Universal Robots PolyScope program: Assignment.urp

Program Assignment (installation=assignment directory=/home/mtrn4230/ursim-5.10.0.106288/programs createdIn=5.10.0.106288 lastSavedIn=5.10.0.106288 robotSerialNumber=20195599999)
Calibrated DH parameters: a=[0, -0.425, -0.3922, 0, 0, 0]; d=[0.1625, 0, 0, 0.1333, 0.0997, 0.0996]; alpha=[1.570796, 0, 0, 1.570796, -1.570796, 0]; deltaTheta=[0, 0, 0, 0, 0, 0]
Robot Program (runOnlyOnce=false)
  SuppressedNode
    Popup Message (haltProgram=false message=EDLYN LIEW L inputType=Text)
  LETTERS := [5,4,13,25,14,27,12,9,5,23,27,12]
  num_letters := 12
  counter := 0
  MoveJ speed 60 deg/s, acceleration 80 deg/s^2 (useActiveTCP=true) feature=letter_start
    Waypoint start_corner: TCP in base x=-509.831 y=-90.3 z=70 mm, rx=2.2214 ry=2.2214 rz=0 rad; joints [-4.875, -57.642, 121.444, -153.801, -90, -4.875] deg; feature pose in base x=-509.831 y=-90.3 z=70 mm, rx=2.2214 ry=2.2214 rz=0 rad
    'start height: 70mm'
  MoveJ speed 60 deg/s, acceleration 80 deg/s^2 (useActiveTCP=true) feature=letter_start
    curr_pos := pose_trans(pose_sub(get_actual_tcp_pose(),letter_start), p[0,0,0,0,0,0])
    Loop While (checkContinuously=false) expression=counter<num_letters
      Switch expression=LETTERS[counter]
        Case (caseValue=1)
          'a'
        Case (caseValue=2)
          'b'
        Case (caseValue=3)
          'c'
        Case (caseValue=4)
          'd'
          Wait Sleep waitTime=1
          MoveJ speed 60 deg/s, acceleration 80 deg/s^2 (useActiveTCP=true) feature=letter_start
            curr_pos := pose_trans(curr_pos, p[0.65/100,0,0,0,0,0])
            Popup Message (haltProgram=false inputType=Variable) variable=curr_pos
            Waypoint Waypoint (Variable): variable=curr_pos
          MoveL speed 250 mm/s, acceleration 1200 mm/s^2 (useActiveTCP=true) feature=letter_start
            Call move_down
            curr_pos := pose_trans(curr_pos, p[0,2/100,0,0,0,0])
            Popup Message (haltProgram=false inputType=Variable) variable=curr_pos
            Waypoint Waypoint (Variable): variable=curr_pos
            end_circle := curr_pos
            Popup Message (haltProgram=false inputType=Variable) variable=curr_pos
            Call move_up
            curr_pos := pose_trans(curr_pos, p[0,-2/100,0,0,0,0])
            Call move_down
            Popup Message (haltProgram=false inputType=Variable) variable=curr_pos
          MoveP speed 250 mm/s, acceleration 1200 mm/s^2 (blendRadius=0.025 useActiveTCP=true) feature=letter_start
            Waypoint Waypoint (Variable): variable=curr_pos
            circle_via := pose_trans(curr_pos, p[1.35/100,1/100,0,0,0,0])
            CircleMove (OrientationMode=UNCONSTRAINED)
              Waypoint Waypoint (Variable): variable=circle_via
              Waypoint Waypoint (Variable): variable=end_circle
          MoveL speed 250 mm/s, acceleration 1200 mm/s^2 (useActiveTCP=true) feature=letter_start
            curr_pos := end_circle
            Waypoint Waypoint (Variable): variable=curr_pos
            Call move_up
            curr_pos := pose_trans(curr_pos, p[1.35/100,-2/100,0,0,0,0])
        Case (caseValue=5)
          'e'
          Wait Sleep waitTime=1
          MoveL speed 250 mm/s, acceleration 1200 mm/s^2 (useActiveTCP=true) feature=letter_start
            Call move_down
            curr_pos := pose_trans(curr_pos, p[0,2/100,0,0,0,0])
            Waypoint Waypoint (Variable): variable=curr_pos
            SuppressedNode
              Popup Message (haltProgram=false inputType=Variable) variable=curr_pos
            curr_pos := pose_trans(curr_pos, p[1/100,0,0,0,0,0])
            SuppressedNode
              Popup Message (haltProgram=false inputType=Variable) variable=curr_pos
            Waypoint Waypoint (Variable): variable=curr_pos
            Call move_up
            SuppressedNode
              Popup Message (haltProgram=false inputType=Variable) variable=curr_pos
            curr_pos := pose_trans( curr_pos,p[-1/100,-2/100,0,0,0,0])
            SuppressedNode
              Popup Message (haltProgram=false inputType=Variable) variable=curr_pos
            Waypoint Waypoint (Variable): variable=curr_pos
            Call move_down
            curr_pos := pose_trans(curr_pos, p[1.1/100,0,0,0,0,0])
            Waypoint Waypoint (Variable): variable=curr_pos
            Call move_up
            curr_pos := pose_trans(curr_pos,p[-1.1/100,0.9/100,0,0,0,0])
            Waypoint Waypoint (Variable): variable=curr_pos
            Call move_down
            curr_pos := pose_trans(curr_pos, p[1/100,0,0,0,0,0])
            Waypoint Waypoint (Variable): variable=curr_pos
            Popup Message (haltProgram=false inputType=Variable) variable=curr_pos
            Call move_up
            curr_pos := pose_trans(curr_pos, p[0.1/100,-0.9/100,0,0,0,0])
            Waypoint Waypoint (Variable): variable=curr_pos
            Popup Message (haltProgram=false inputType=Variable) variable=curr_pos
        Case (caseValue=6)
          'f'
        Case (caseValue=7)
          'g'
        Case (caseValue=8)
          'h'
        Case (caseValue=9)
          'i'
        Case (caseValue=10)
          'j'
        Case (caseValue=11)
          'k'
        Case (caseValue=12)
          'l'
          Wait Sleep waitTime=1
          MoveL speed 250 mm/s, acceleration 1200 mm/s^2 (useActiveTCP=true) feature=letter_start
            curr_pos := pose_trans(curr_pos, p[0.7/100,0,0,0,0,0])
            Waypoint Waypoint (Variable): variable=curr_pos
            Call move_down
            curr_pos := pose_trans(curr_pos, p[0,2/100,0,0,0,0])
            Waypoint Waypoint (Variable): variable=curr_pos
            curr_pos := pose_trans(curr_pos, p[1/100,0,0,0,0,0])
            Waypoint Waypoint (Variable): variable=curr_pos
            Call move_up
            curr_pos := pose_trans(curr_pos,p[0.2/100,-2/100,0,0,0,0])
        Case (caseValue=13)
          'm'
        Case (caseValue=14)
          'n'
          Wait Sleep waitTime=1
          MoveJ speed 60 deg/s, acceleration 80 deg/s^2 (useActiveTCP=true) feature=letter_start
            curr_pos := pose_trans(curr_pos, p[0.3,0,0,0,0,0])
            Waypoint Waypoint (Variable): variable=curr_pos
            Call move_down
            curr_pos := pose_trans(curr_pos, p[0,2/100,0,0,0,0])
            Waypoint Waypoint (Variable): variable=curr_pos
            Call move_up
            curr_pos := pose_trans(curr_pos, p[0,-2/100,0,0,0,0])
            Waypoint Waypoint (Variable): variable=curr_pos
            Call move_down
            curr_pos := pose_trans(curr_pos, p[1.25/100,2/100,0,0,0,0])
            Waypoint Waypoint (Variable): variable=curr_pos
            Call move_up
            curr_pos := pose_trans(curr_pos, p[0,-2/100,0,0,0,0])
            Waypoint Waypoint (Variable): variable=curr_pos
            Call move_down
            curr_pos := pose_trans(curr_pos, p[0,2/100,0,0,0,0])
            Waypoint Waypoint (Variable): variable=curr_pos
            Call move_up
            curr_pos := pose_trans(curr_pos, p[0.2/100,-2/100,0,0,0,0])
        Case (caseValue=15)
          'o'
        Case (caseValue=16)
          'p'
        Case (caseValue=17)
          'q'
        Case (caseValue=18)
          'r'
        Case (caseValue=19)
          's'
        Case (caseValue=20)
          't'
        Case (caseValue=21)
          'u'
        Case (caseValue=22)
          'v'
        Case (caseValue=23)
          'w'
        Case (caseValue=24)
          'x'
        Case (caseValue=25)
          'y'
          Wait Sleep waitTime=1
          MoveJ speed 60 deg/s, acceleration 80 deg/s^2 (useActiveTCP=true) feature=letter_start
            curr_pos := pose_trans(curr_pos, p[0.3/100,0,0,0,0,0])
            Waypoint Waypoint (Variable): variable=curr_pos
            Call move_down
            curr_pos := pose_trans(curr_pos, p[0.8/100,1.3/100,0,0,0,0])
            Waypoint Waypoint (Variable): variable=curr_pos
            Call move_up
            curr_pos := pose_trans(curr_pos, p[0.8/100,-1.3/100,0,0,0,0])
            Waypoint Waypoint (Variable): variable=curr_pos
            Call move_down
            curr_pos := pose_trans(curr_pos, p[-0.8/100,1.3/100,0,0,0,0])
            Waypoint Waypoint (Variable): variable=curr_pos
            curr_pos := pose_trans(curr_pos, p[0,0.8/100,0,0,0,0])
            Waypoint Waypoint (Variable): variable=curr_pos
            Call move_up
            curr_pos := pose_trans(curr_pos, p[1/100,-2/100,0,0,0,0])
        Case (caseValue=26)
          'z'
        Case (caseValue=27)
          'space'
          Wait Sleep waitTime=1
          curr_pos := pose_trans(curr_pos, p[2.2/100,0,0,0,0,0])
      counter := counter+1
  MoveJ speed 60 deg/s, acceleration 80 deg/s^2 (useActiveTCP=true) feature=letter_start
    Waypoint start_corner: TCP in base x=-509.831 y=-90.3 z=70 mm, rx=2.2214 ry=2.2214 rz=0 rad; joints [-4.875, -57.642, 121.444, -153.801, -90, -4.875] deg
  Popup Message (haltProgram=true message=Program completed inputType=Text)
  URCap External Control (External Control, FZI Research Center for Information Technology)
SubProgram -> move_up
SubProgram -> move_down
SubProgram move_down (keepSynchronizedWithDisk=false) programFile=/home/mtrn4230/ursim-5.10.0.106288/programs/move down.urp
  MoveL speed 250 mm/s, acceleration 1200 mm/s^2 (useActiveTCP=true) feature=letter_start
    curr_pos := pose_add(curr_pos, p[0,0,1/100,0,0,0])
    Waypoint Waypoint (Variable): variable=curr_pos
SubProgram move_up (keepSynchronizedWithDisk=false) programFile=/home/mtrn4230/ursim-5.10.0.106288/programs/move up.urp
  MoveL speed 250 mm/s, acceleration 1200 mm/s^2 (useActiveTCP=true) feature=letter_start
    curr_pos := pose_add(curr_pos, p[0,0,-1/100,0,0,0])
    Waypoint Waypoint (Variable): variable=curr_pos
